FUNCTION_BLOCK T_CartesianRobot EXTENDS T_NamedBase
VAR
	_xAxis, _yAxis, _zAxis : I_Axis;
	_gripper : I_Gripper;
END_VAR

METHOD GenericInitialise : BOOL;
VAR_INPUT
	xAxis, yAxis, zAxis : I_Axis;
	gripper : I_Gripper;
END_VAR
IF xAxis = 0 OR yAxis = 0 OR yAxis = 0 OR gripper = 0 THEN
    RETURN;
END_IF

_xAxis := xAxis;
_yAxis := yAxis;
_zAxis := zAxis;
_gripper := gripper;

GenericInitialise := TRUE;
END_METHOD

END_FUNCTION_BLOCK

(* stored: Version 1.1.0.1, ProductVersion 3.1.4024.12
   POU T_CartesianRobot: Id {2f13929b-38b0-4c49-93c6-1008e6f60238}, SpecialFunc None
   Method GenericInitialise: Id {7c60b10c-ac22-43b1-bb25-35dbf1d96bf3} *)
